FUNCTION_BLOCK PoweredStatus
VAR_INPUT
	///Super state (TRUE if the super state is active, or if there is no super state)
	superState: BOOL := TRUE;
	///TRUE if power is enabled
	isEnabled: BOOL;
END_VAR
VAR_OUTPUT
	///The power is enabled
	{attribute 'OPC.UA.DA' := '1'}
	{attribute 'OPC.UA.DA.Access' := '1'}
	enabled: BOOL;
	///The power is disabled
	{attribute 'OPC.UA.DA' := '1'}
	{attribute 'OPC.UA.DA.Access' := '1'}
	disabled: BOOL;
END_VAR
VAR_IN_OUT
END_VAR
VAR
END_VAR

enabled := isEnabled AND superState;
disabled := (NOT(isEnabled)) AND superState;

END_FUNCTION_BLOCK

(* stored: Version 1.1.0.1, ProductVersion 3.1.4019.2
   POU PoweredStatus: Id {a319f636-a232-476e-bb98-5526862376f9}, SpecialFunc None *)
